(****************************************************************
NAME:			FB_SetAxisPosition
DATA:			2017.2.16
VERSION:		1.0.0
DESCRIPTION:	FB_SetAxisPosition
HISTORY:
				2017.2.16		NEW

***************************************************************)
FUNCTION_BLOCK FB_SetAxisPosition
VAR_INPUT
	//GapValueSet:LREAL:=0;
	ValueSet_LeftTop:LREAL:=0;
	ValueSet_RightTop:LREAL:=0;
	ValueSet_LeftBottom:LREAL:=0;
	ValueSet_RightBottom:LREAL:=0;
	ValueSet_LeftIn:LREAL:=0;
	ValueSet_RightIn:LREAL:=0;
	ValueSet_LeftOut:LREAL:=0;
	ValueSet_RightOut:LREAL:=0;
	Execute:BOOL;
END_VAR
VAR_OUTPUT
	FbID:DINT:=1001;
	State:DINT;
	Busy:BOOL;
	Done:BOOL;
	Error:BOOL;
	ErrorID:DINT;
END_VAR
VAR
	LeftTopLin_MC_SetPosition: MC_SetPosition;
	RightTopLin_MC_SetPosition: MC_SetPosition;
	LeftBottomLin_MC_SetPosition: MC_SetPosition;
	RightBottomLin_MC_SetPosition: MC_SetPosition;
	LeftInLin_MC_SetPosition: MC_SetPosition;
	RightInLin_MC_SetPosition: MC_SetPosition;
	LeftOutLin_MC_SetPosition: MC_SetPosition;
	RightOutLin_MC_SetPosition: MC_SetPosition;
	fb_ton: TON;
	FB_PlcEmergencyStop: FB_PlcEmergencyStop;

END_VAR

IF Execute THEN
Busy:=TRUE;
Done:=FALSE;
fb_ton(PT:=t#0.1s);
CASE State OF
	0:
		IF LeftTopLin_MC_SetPosition.Error OR RightTopLin_MC_SetPosition.Error
			OR LeftBottomLin_MC_SetPosition.Error OR RightBottomLin_MC_SetPosition.Error 
			OR LeftInLin_MC_SetPosition.Error OR RightInLin_MC_SetPosition.Error
			OR LeftOutLin_MC_SetPosition.Error OR RightOutLin_MC_SetPosition.Error THEN		(*FB Error*)
			ErrorID:=1;
			State:=99;
		ELSE
			State:=1;
		END_IF
	1:	(*Execute*)
		LeftTopLin_MC_SetPosition.Position:=ValueSet_LeftTop;
		LeftTopLin_MC_SetPosition.Execute:=TRUE;
		RightTopLin_MC_SetPosition.Position:=ValueSet_RightTop;
		RightTopLin_MC_SetPosition.Execute:=TRUE;
		LeftBottomLin_MC_SetPosition.Position:=ValueSet_LeftBottom;
		LeftBottomLin_MC_SetPosition.Execute:=TRUE;
		RightBottomLin_MC_SetPosition.Position:=ValueSet_RightBottom;
		RightBottomLin_MC_SetPosition.Execute:=TRUE;
		//
		LeftInLin_MC_SetPosition.Position:=ValueSet_LeftIn;
		LeftInLin_MC_SetPosition.Execute:=TRUE;
		RightInLin_MC_SetPosition.Position:=ValueSet_RightIn;
		RightInLin_MC_SetPosition.Execute:=TRUE;
		LeftOutLin_MC_SetPosition.Position:=ValueSet_LeftOut;
		LeftOutLin_MC_SetPosition.Execute:=TRUE;
		RightOutLin_MC_SetPosition.Position:=ValueSet_RightOut;
		RightOutLin_MC_SetPosition.Execute:=TRUE;
		A_SetPositionMC();
		fb_ton.IN:=TRUE;
		State:=2;
	2:	(*Wait*)
		A_SetPositionMC();
		IF NOT LeftTopLin_MC_SetPosition.Done OR NOT RightTopLin_MC_SetPosition.Done
			OR NOT LeftBottomLin_MC_SetPosition.Done OR NOT RightBottomLin_MC_SetPosition.Done 
			OR NOT LeftInLin_MC_SetPosition.Done OR NOT RightInLin_MC_SetPosition.Done
			OR NOT LeftOutLin_MC_SetPosition.Done OR NOT RightOutLin_MC_SetPosition.Done THEN		(*DoneÐÅºÅ²»µ½£¬¼ÌÐøµÈ´ý£¬Èç¹û³¬Ê±ÔòFB Error*)
			IF NOT fb_ton.Q THEN
				State:=2;
			ELSE
				ErrorID:=4;
				State:=99;
			END_IF
		ELSIF  LeftTopLin_MC_SetPosition.Done AND RightTopLin_MC_SetPosition.Done
			AND LeftBottomLin_MC_SetPosition.Done AND RightBottomLin_MC_SetPosition.Done 
			AND LeftInLin_MC_SetPosition.Done AND RightInLin_MC_SetPosition.Done
			AND LeftOutLin_MC_SetPosition.Done AND RightOutLin_MC_SetPosition.Done THEN		(*Done£¬×ªÏÂÒ»²½*)
			State:=88;
		ELSE
			ErrorID:=5;
			State:=99;
		END_IF
	88:
		Execute:=FALSE;
		State:=0;
		Busy:=FALSE;
		Done:=TRUE;
		Error:=FALSE;
		ErrorID:=0;
		LeftTopLin_MC_SetPosition.Execute:=FALSE;
		RightTopLin_MC_SetPosition.Execute:=FALSE;
		LeftBottomLin_MC_SetPosition.Execute:=FALSE;
		RightBottomLin_MC_SetPosition.Execute:=FALSE;
		LeftInLin_MC_SetPosition.Execute:=FALSE;
		RightInLin_MC_SetPosition.Execute:=FALSE;
		LeftOutLin_MC_SetPosition.Execute:=FALSE;
		RightOutLin_MC_SetPosition.Execute:=FALSE;
		fb_ton.IN:=FALSE;
	99:
		Execute:=FALSE;
		State:=99;
		Busy:=FALSE;
		Done:=FALSE;
		Error:=TRUE;
		LeftTopLin_MC_SetPosition.Execute:=FALSE;
		RightTopLin_MC_SetPosition.Execute:=FALSE;
		LeftBottomLin_MC_SetPosition.Execute:=FALSE;
		RightBottomLin_MC_SetPosition.Execute:=FALSE;
		LeftInLin_MC_SetPosition.Execute:=FALSE;
		RightInLin_MC_SetPosition.Execute:=FALSE;
		LeftOutLin_MC_SetPosition.Execute:=FALSE;
		RightOutLin_MC_SetPosition.Execute:=FALSE;
		fb_ton.IN:=FALSE;
	-100:
		FB_PlcEmergencyStop();
		Execute:=FALSE;
		State:=-100;
		Busy:=FALSE;
		Done:=FALSE;
		Error:=TRUE;
		LeftTopLin_MC_SetPosition.Execute:=FALSE;
		RightTopLin_MC_SetPosition.Execute:=FALSE;
		LeftBottomLin_MC_SetPosition.Execute:=FALSE;
		RightBottomLin_MC_SetPosition.Execute:=FALSE;
		
		LeftInLin_MC_SetPosition.Execute:=FALSE;
		RightInLin_MC_SetPosition.Execute:=FALSE;
		LeftOutLin_MC_SetPosition.Execute:=FALSE;
		RightOutLin_MC_SetPosition.Execute:=FALSE;
		fb_ton.IN:=FALSE;
END_CASE
END_IF

ACTION A_SetPositionMC:
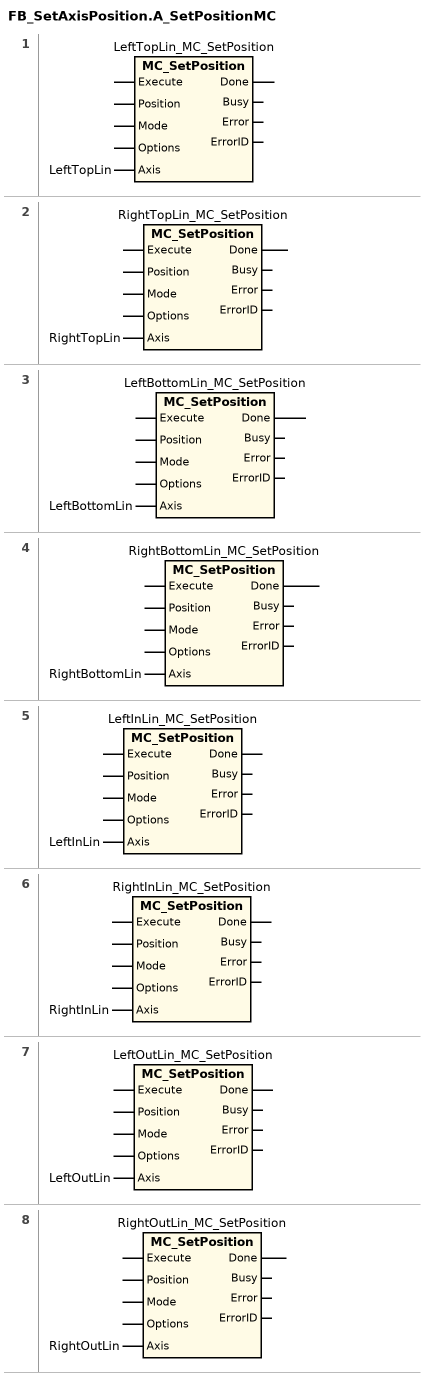
// NETWORK 1
LeftTopLin_MC_SetPosition(Axis := LeftTopLin); // MC_SetPosition

// NETWORK 2
RightTopLin_MC_SetPosition(Axis := RightTopLin); // MC_SetPosition

// NETWORK 3
LeftBottomLin_MC_SetPosition(Axis := LeftBottomLin); // MC_SetPosition

// NETWORK 4
RightBottomLin_MC_SetPosition(Axis := RightBottomLin); // MC_SetPosition

// NETWORK 5
LeftInLin_MC_SetPosition(Axis := LeftInLin); // MC_SetPosition

// NETWORK 6
RightInLin_MC_SetPosition(Axis := RightInLin); // MC_SetPosition

// NETWORK 7
LeftOutLin_MC_SetPosition(Axis := LeftOutLin); // MC_SetPosition

// NETWORK 8
RightOutLin_MC_SetPosition(Axis := RightOutLin); // MC_SetPosition
END_ACTION

END_FUNCTION_BLOCK

(* stored: Version 1.1.0.1, ProductVersion 3.1.4024.6
   POU FB_SetAxisPosition: Id {6afa31ff-e0ae-4621-979a-f7f274bb3d8a}, SpecialFunc None
   Action A_SetPositionMC: Id {9afeaa97-7af6-44a0-91c2-9bb3ac449bed} *)
